TYPE ST_SettingsUnlockingPins :
STRUCT
	tPinsLockTimeout : TIME := T#10S;	/// Timeout for locking pins [default: 10s]
	tPinsUnlockTimeout : TIME := T#10S;	/// Timeout for unlocking pins [default: 10s]
END_STRUCT
END_TYPE

(* stored: Version 1.1.0.1, ProductVersion 3.1.4024.12
   DUT ST_SettingsUnlockingPins: Id {41d564fd-bb6d-44f6-a928-3276c82e112b} *)
